{attribute addProperty BoxType "EL2212-0000-0018"}
{attribute addProperty Id "Ready_to_activateBIT10.1251Output_activeBIT10.1252Tristate_activeBIT10.1253WarningBIT10.1257ErrorBIT10.1258Sync_errorBIT10.12514TxPDO_ToggleBIT10.12516"}
{attribute addProperty CRC "1568505292"}
{attribute addProperty SizeInBites "16"}
{attribute addProperty SizeInBytes "2"}
TYPE Status_5D7D7DCC :
STRUCT
	{attribute addProperty Name "Ready_to_activate"}
	Ready_to_activate : BIT;
	{attribute addProperty Name "Output_active"}
	Output_active : BIT;
	{attribute addProperty Name "Tristate_active"}
	Tristate_active : BIT;
	{attribute 'hide'}
	reserve_1_BIT_0 : BIT;
	{attribute 'hide'}
	reserve_1_BIT_1 : BIT;
	{attribute 'hide'}
	reserve_1_BIT_2 : BIT;
	{attribute addProperty Name "Warning"}
	Warning : BIT;
	{attribute addProperty Name "Error"}
	Error : BIT;
	{attribute 'hide'}
	reserve_2_BIT_0 : BIT;
	{attribute 'hide'}
	reserve_2_BIT_1 : BIT;
	{attribute 'hide'}
	reserve_2_BIT_2 : BIT;
	{attribute 'hide'}
	reserve_2_BIT_3 : BIT;
	{attribute 'hide'}
	reserve_2_BIT_4 : BIT;
	{attribute addProperty Name "Sync_error"}
	Sync_error : BIT;
	{attribute 'hide'}
	reserve_3 : BIT;
	{attribute addProperty Name "TxPDO_Toggle"}
	TxPDO_Toggle : BIT;
END_STRUCT
END_TYPE

(* stored: Version 1.2.0.0, ProductVersion 3.1.4024.9
   DUT Status_5D7D7DCC: Id {fbc840aa-5ca2-4fe5-98d3-44bb33446c92} *)
